INTERFACE I_Device

END_INTERFACE

(* stored: Version 1.1.0.1, ProductVersion 3.1.4024.12
   Itf I_Device: Id {11111111-2222-3333-4444-555555555555} *)
